// Brief: Slave Arm Adjust
FUNCTION_BLOCK PUBLIC FB_SlaveCtrlAdjust EXTENDS FB_SlaveArmCtrlBase
VAR
	// velocity for full damping
	m_maxAdjustVel :Vec3d := [1.2, 1.2, 0.3];
	
	// velocity start to enable damping
	m_velLBForDamp :Vec3d := [0.7, 0.7, 0.1];
	
	// max damp
	m_maxDamp :Vec3d := [1,1,100];//50, 50, 500
	
	// distance buffer from joint limit to start damp
	m_limitBufferForDamp :Vec3d :=[20*g_deg2Rad, 20*g_deg2Rad, 0.03];
	
	// joint velocity threshold for coulomb friction transition
	m_cFrictionVelThres : LREAL := 5.0 * g_deg2Rad;
	m_frictionCompScale :LREAL :=0.1;
	
	m_forceKp:Vec3d := [1000,1000,2500];
	m_forceKv:Vec3d := [100,100,150];
	m_upLimit:Vec3d :=g_zeroVec3d;
	m_lowLimit:Vec3d :=g_zeroVec3d;
END_VAR

// override this function in each exact controller
METHOD PROTECTED calcCmdJntPos : BOOL
VAR_IN_OUT CONSTANT
	i_endoscopePose : ST_Frame;
	i_masterStatus :ST_MasterStatus;
	i_setupStatus: ST_SetupStatus;
	i_slaveArm :FB_SlaveArm;
END_VAR
VAR
	i:INT;
END_VAR
FOR i:= 1 TO 8 DO
	IF m_jntOPMode[i] = DriverOPMode_Trq THEN
		m_cmdJntPos[i]:=i_slaveArm.curJntPos[i];
	END_IF
END_FOR

m_cmdCartPose:=i_slaveArm.curCartPose;
END_METHOD

// override this function in each exact controller
METHOD PROTECTED calcCmdJntTrq : BOOL
VAR_IN_OUT CONSTANT
	i_endoscopePose : ST_Frame;
	i_masterStatus :ST_MasterStatus;
	i_setupStatus: ST_SetupStatus;
	i_slaveArm :FB_SlaveArm;
END_VAR
VAR
	i :INT;
	dampScale :LREAL;
	limitDis:LREAL;
	transitScale:LREAL;
	cFriction:LREAL;
	limitTrq:LREAL;
END_VAR
// set joint torque to zero in default
m_cmdJntTrq := g_zeroVec8d;

// disable joints if this joint is an unrecoverable failure
FOR i:=1 TO g_sJntNum DO
	IF SafetyCheck.m_SafetyCheck.m_jntErrFlag[i_slaveArm.armIdx, 0, 3] OR  SafetyCheck.m_SafetyCheck.m_jntErrFlag[i_slaveArm.armIdx, i+g_setupJntNum, 3] THEN
		m_jntEnableFlag[i] := 0;
	ELSE
		m_jntEnableFlag[i] := 1;
	END_IF
END_FOR

// enable endoscope rotation joint if external torque exceed specific value
IF i_slaveArm.instrument.onChipData.m_InstruReadSucceed AND i_slaveArm.instrument.instruType = InstruType_Endoscope THEN
		FOR i:=6 TO 8 DO 
			IF ABS(i_slaveArm.filtJntCurrent[i]) > 100 THEN
				m_jntOPMode[i]:=DriverOPMode_Trq;
			END_IF
		END_FOR
END_IF

// add joint limit constraint
FOR i:=1 TO 3 DO
	m_upLimit[i]:= MAX(GVL_SlaveMotorParameters.g_maxDHJntPos[i], MIN(m_upLimit[i], i_slaveArm.curJntPos[i]));
	m_lowLimit[i]:= MIN(GVL_SlaveMotorParameters.g_minDHJntPos[i], MAX(m_lowLimit[i], i_slaveArm.curJntPos[i]));

	IF i_slaveArm.curJntPos[i] > m_upLimit[i] THEN
		limitTrq := m_forceKp[i] * (m_upLimit[i]-i_slaveArm.curJntPos[i]) - m_forceKv[i]* i_slaveArm.curJntVel[i];
		m_cmdJntTrq[i] := m_cmdJntTrq[i] + limitTrq;		
	ELSIF i_slaveArm.curJntPos[i] < m_lowLimit[i] THEN
		limitTrq := m_forceKp[i] * (m_lowLimit[i]-i_slaveArm.curJntPos[i]) - m_forceKv[i]* i_slaveArm.curJntVel[i];
		m_cmdJntTrq[i] := m_cmdJntTrq[i] + limitTrq;
	END_IF
END_FOR

// compute damp
FOR i:=1 TO 3 DO
	IF ABS(i_slaveArm.curJntVel[i]) > m_velLBForDamp[i] THEN 
		dampScale:=LIMIT(0, (ABS(i_slaveArm.curJntVel[i])- m_velLBForDamp[i])/(m_maxAdjustVel[i] - m_velLBForDamp[i]), 1 );
		m_cmdJntTrq[i] :=m_cmdJntTrq[i] -i_slaveArm.curJntVel[i] * m_maxDamp[i] * dampScale;
	END_IF
END_FOR

//add friction compensation for joint4
FOR i:=1 TO 2 DO
	transitScale := LIMIT(0, ABS(i_slaveArm.curJntVel[i]/m_cFrictionVelThres),1);
	cFriction:= transitScale * sign(i_slaveArm.curJntVel[i]) * GVL_SlaveArmDynamics.g_slaveJntFriction[i_slaveArm.armIdx,i];
	m_cmdJntTrq[i]:= m_cmdJntTrq[i]+m_frictionCompScale*cFriction;
END_FOR
END_METHOD

METHOD PUBLIC init : BOOL
VAR_IN_OUT CONSTANT
	i_slaveArm	:FB_SlaveArm;
END_VAR
VAR_IN_OUT 
	r_slaveArmCtrlCmd :ST_SlaveArmCtrlCmds;
END_VAR
VAR
	i :INT;
END_VAR
// check if to hold the command joint position unchanged
m_holdLastCmds := checkToHoldLastCmds(i_slaveArm);

//init
SUPER^.Init(i_slaveArm,r_slaveArmCtrlCmd);

// disable joints if this joint is an unrecoverable failure
FOR i:=1 TO g_sJntNum DO
	IF SafetyCheck.m_SafetyCheck.m_jntErrFlag[i_slaveArm.armIdx, 0, 3] OR  SafetyCheck.m_SafetyCheck.m_jntErrFlag[i_slaveArm.armIdx, i+g_setupJntNum, 3] THEN
		m_jntEnableFlag[i] := 0;
	ELSE
		m_jntEnableFlag[i] := 1;
	END_IF
END_FOR

// joint 1/2/3/7 run in torque mode
m_jntOPMode[1]:=DriverOPMode_Trq;
m_jntOPMode[2]:=DriverOPMode_Trq;
m_jntOPMode[3]:=DriverOPMode_Trq;

m_jntOPMode[4]:=DriverOPMode_PosTrq;
m_jntOPMode[5]:=DriverOPMode_PosTrq;
m_jntOPMode[6]:=DriverOPMode_PosTrq;
m_jntOPMode[7]:=DriverOPMode_PosTrq;
m_jntOPMode[8]:=DriverOPMode_PosTrq;

IF i_slaveArm.instrument.onChipData.m_InstruReadSucceed THEN
	IF i_slaveArm.instrument.instruType <> InstruType_Endoscope THEN
		m_jntOPMode[7]:=DriverOPMode_Trq;
	END_IF
END_IF

// hold joint3 if instrument mount failed
IF i_slaveArm.instruOn AND NOT(SlaveArmControl.m_slaveRobot.m_instrumentMountedFlag[i_slaveArm.armIdx]) THEN
	m_jntOPMode[3]:=DriverOPMode_PosTrq;
END_IF

FOR i:=1 TO 3 DO
	m_upLimit[i]:= MAX(GVL_SlaveMotorParameters.g_maxDHJntPos[i], i_slaveArm.curJntPos[i]);
	m_lowLimit[i]:= MIN(GVL_SlaveMotorParameters.g_minDHJntPos[i], i_slaveArm.curJntPos[i]);
END_FOR

// update commands to arm
copyCmds(r_slaveArmCtrlCmd);
END_METHOD

END_FUNCTION_BLOCK

(* stored: Version 1.1.0.1, ProductVersion 3.1.4024.11
   POU FB_SlaveCtrlAdjust: Id {065dc40e-4d51-49bc-8f28-94a80cbbd0fd}, SpecialFunc None
   Method calcCmdJntPos: Id {702c20a9-7bcc-49ed-9f8d-b2e61f393510}
   Method calcCmdJntTrq: Id {fcf0acdf-cfca-4de6-b628-f0f18f7171ce}
   Method init: Id {0b0d07b9-f0c8-4405-b76e-2338c9ecb922} *)
